TYPE typeSetupMachine :
STRUCT
	
//stations
stationFunctions: ARRAY[1..gHMIDataConsts.gNumberOfStations] OF typeSetupStation;
stationEnable: ARRAY[1..gHMIDataConsts.gNumberOfStations] OF BOOL;



END_STRUCT
END_TYPE

(* stored: Version 1.1.0.1, ProductVersion 3.1.4024.12
   DUT typeSetupMachine: Id {d75b749f-7d0d-4c7b-8cf0-880ec94762fe} *)
